{attribute addProperty BoxType "EJ7342-0000-0019"}
{attribute addProperty Id "StatusAT %I*Status_1C57BC2B162"}
{attribute addProperty CRC "3266366177"}
{attribute addProperty SizeInBites "16"}
{attribute addProperty SizeInBytes "2"}
TYPE DCM_Status_Channel_C2B0CAE1 :
STRUCT
	{attribute addProperty Name "Status"}
	Status AT %I* : Status_1C57BC2B;
END_STRUCT
END_TYPE

(* stored: Version 1.2.0.0, ProductVersion 3.1.4024.9
   DUT DCM_Status_Channel_C2B0CAE1: Id {50d7e0d4-9c94-4209-9ef4-38c752e2398b} *)
